SUBAPPLICATION mapping_Uebung_036 (* Spiegelabfolge V2 mit Schrittkette *)
  (* Standard: 61499-2; Description: Copyright (c) 2023 Meisterschulen am Ostbahnhof This program and the accompanying materials are made available under the terms of the Eclipse Public License 2.0 which is available at https://www.eclipse.org/legal/epl-2.0/ SPDX-License-Identifier: EPL-2.0 *)
  (* Version 1.0, 2023-10-23, Franz Höpfinger, Meisterschulen am Ostbahnhof *)
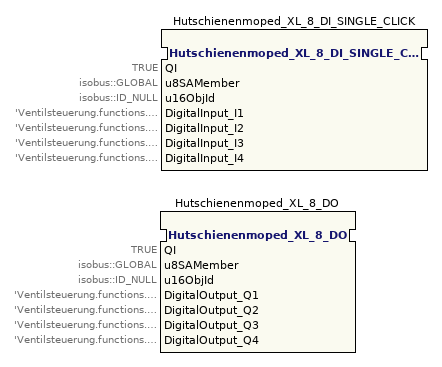
  FBS
    Hutschienenmoped_XL_8_DO : Hutschienenmoped_XL_8_DO(QI := TRUE, u8SAMember := isobus::GLOBAL, u16ObjId := isobus::ID_NULL, DigitalOutput_Q1 := 'Ventilsteuerung.functions.DigitalOutput_Q1', DigitalOutput_Q2 := 'Ventilsteuerung.functions.DigitalOutput_Q2', DigitalOutput_Q3 := 'Ventilsteuerung.functions.DigitalOutput_Q3', DigitalOutput_Q4 := 'Ventilsteuerung.functions.DigitalOutput_Q4');
    Hutschienenmoped_XL_8_DI_SINGLE_CLICK : Hutschienenmoped_XL_8_DI_SINGLE_CLICK(QI := TRUE, u8SAMember := isobus::GLOBAL, u16ObjId := isobus::ID_NULL, DigitalInput_I1 := 'Ventilsteuerung.functions.DigitalInput_CLK_I1', DigitalInput_I2 := 'Ventilsteuerung.functions.DigitalInput_CLK_I2', DigitalInput_I3 := 'Ventilsteuerung.functions.DigitalInput_CLK_I3', DigitalInput_I4 := 'Ventilsteuerung.functions.DigitalInput_CLK_I4');
  END_FBS
END_SUBAPPLICATION
